Fanuc KAREL source: kt00530.KL

-- PROVISIONAL review KL for V1013-1; original PC SHA256 d1561f2aca54913408bacf8fa10a6fd8ddf6001ee17d7d5694babaabf23933e5
-- Incomplete behavior may be omitted. Consult companion uncertainty JSON. Do not deploy.
PROGRAM KT00530
%NOLOCKGROUP
-- UNRESOLVED_DECL P1 type=000106
-- UNRESOLVED_DECL P2 type=000199
-- UNRESOLVED_DECL OUT type=000102
BEGIN
  -- UNRESOLVED_PC offsets 5-20; opcodes 2E,22,32,35
  -- UNRESOLVED_PC offsets 25-64; opcodes 49,7E,49,7E,60,7E,4A
  -- UNRESOLVED_PC offsets 69-73; opcodes 7F
END KT00530
